# EPICS autosave request: iocBoot/sioc-esb-sint01/softInt.req
file ../common.req P=$(P), N=01
